(* IEC 61131-3 sources: verifaps-lib/geteta/examples/issue5, 1 file *)

(* ---- issue5.st ---- *)
PROGRAM var_GetetaOffByOne

  VAR_OUTPUT
    var_counter  : INT  := 0;
  END_VAR

  var_counter := var_counter + 1;

END_PROGRAM
